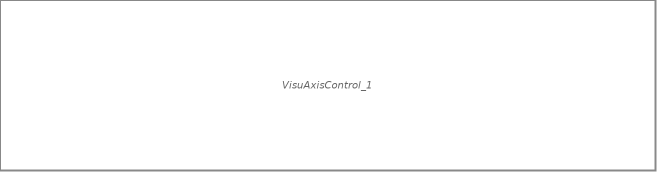
VISUALIZATION VisuAxisX_1  // 657x172
    Frame (0,0 655x170)
        shows VisuAxisControl_1(sAxisName_1 := sAxisXName, stAxisVisu_1 := stAxisX)
END_VISUALIZATION

(* stored: Version 1.1.0.1, ProductVersion 3.1.4022.6
   Visu VisuAxisX_1: Id {6927c8ed-906d-41cc-8934-a474259b710e} *)
